FUNCTION_BLOCK FB_Example
VAR
    Counter : INT;
END_VAR
BEGIN
counter := 1;
END_FUNCTION_BLOCK
